# EPICS substitutions: timingApp/Db/timing.substitutions
file "perStatisticCounter.template"
{ pattern
{       T,               NAME,                         DESC }
  { "\$(T)", InjSeqNoConnectionCount,      "" }
  { "\$(T)", InjSeqStartOverrunCount,      "" }
  { "\$(T)", InjSeqStaleSequenceCount,     "" }
  { "\$(T)", InjSeqInvalidModeCount,       "" }
  { "\$(T)", InjSeqInvalidBucketCount,     "" }
  { "\$(T)", InjSeqInvalidBunchesCount,    "" }
  { "\$(T)", InjSeqNoBeamCurrentCount,     "" }
  { "\$(T)", InjSeqBadBeamCurrentCount,    "" }
  { "\$(T)", InjExcessiveBeamCurrentCount, "" }
  { "\$(T)", InjSeqBadSeverityCount,       "" }
  { "\$(T)", InjSeqBadEVRCount,            "" }
  { "\$(T)", InjSeqSyncDelayTimeoutCount,  "" }
  { "\$(T)", InjSeqSuccessCount,           "" }
  { "\$(T)", InjSeqFailedCount,            "" }
  { "\$(T)", InjSeqDebug,                  "Enable sequencer diagnostic messages" }
}
